FUNCTION F_SignaldauerVonTastleuchte_MaschEinAuswerten : BOOL
VAR_INPUT
END_VAR
VAR
	wTmp : UDINT;
	setPnozSigLen : BOOL := FALSE;
END_VAR

//HIER WEITER
(*      
	  U     "E0_1"
      X     "M 3.1"
      SPBN  s1
*)

setPnozSigLen := FALSE;

IF IO.inResetNotHalt XOR VAT.bResetNotHalt_Old THEN //war M3.1

(*
      U     "E0_1"
      =     "M 3.1"
      SPB   zm
	  *)
	  //VAT.bResetNotHalt_Old := IO.inResetNotHalt; NBT - hier weggenommen...
	  //IF NOT IO.inResetNotHalt THEN
		  (*
		  L     999
		  L     "T 71"	-- gehe davon aus, dass er die Zeit von T71 lädt...
		  -I    		-- AKKU1 von AKKU2 subtrahieren
		  +     -1		-- Ganzzahl addieren
		  L     4
		  /I    		-- AKKU2 durch AKKU1 dividieren
		  L     4		
		  *I    		-- AKKU1 und AKKU2 multiplizieren
		  T     "DB6".w230
		  *)
		  //ToDo, noch keine Ahnung, was das soll...(LSB's verschwinden lassen)
		  //DB6.w230 := 999 - TIME_TO_INT(GVL.tofPnozSigLen.ET);
	  //END_IF
	  (*
zm:   BLD   130
      SET  -- VKE auf 1 setzen (=1)  
      L     S5T#9S990MS
      SA    "T 71" -- Zeit mit Ausschaltverzögerung start vorbereiten mit VKE=1
      CLR   VKE auf 0 setzen 
      SA    "T 71" -- Zeit mit Ausschaltverzögerung starten mit VKE=0
*)
setPnozSigLen := TRUE;
	  
END_IF //of IF IO.e01PNOZ_Signal XOR VAT.M3.1 ...

//GVL.tofPnozSigLen(IN := setPnozSigLen, PT := T#9S990MS); //(ehem. T71)

VAT.bResetNotHalt_Old := IO.inResetNotHalt; //NBT - hier hingesetzt...

(*	  
s1:   BLD   130
      UN    "E0_1"
      L     S5T#1S200MS
      SE    "T 70"
*)
//GVL.tonPnozEntprell(IN := NOT IO.inResetNotHalt, PT := T#1S200MS); //(ehem. T70)
(*	  
      U     "E0_1"
      L     S5T#1S
      SE    "T 72"
*)
//GVL.tonSAFETYok(IN := IO.safeOutHauptLuft, PT := T#1S); -- von hier weg nach P_InputHandling()

END_FUNCTION

(* stored: Version 1.1.0.1, ProductVersion 3.1.4024.3
   POU F_SignaldauerVonTastleuchte_MaschEinAuswerten: Id {8c5f9cd0-205b-47a9-afc3-9a8da24111a4}, SpecialFunc None *)
